// TIA Portal project "12_Converge_Station" (V19)

(* hardware
DEVICE "S7-1500/ET200MP station_1"  S7-1500 station
   slot 0: "Rail_0"  Rack  6ES7 590-1***0-0AA0
   slot 1: "PLC_1"  CPU 1513-1 PN  6ES7 513-1AL02-0AB0  V2.9
      slot 3: "CPU display_1"  6ES7591-1AA00-0AA0
      slot 32768: "PROFINET interface_1"  X1
         slot 32769: "Port_1"  X1 P1
         slot 32770: "Port_2"  X1 P2
      slot 34817: "Virtual CP interface port_1"  Virtual CP interface port  Virtual CP interface port
*)

// ===== PLC "PLC_1"  CPU 1513-1 PN =====

VAR_GLOBAL   // PLC tag table "Default tag table"
   "nw2" AT %M0.0 : Bool;
   "nw3 2nd memory (Pause)" AT %M0.2 : Bool;
   "nw3 1st memory (Unpause)" AT %M0.1 : Bool;
   "nw4" AT %M0.3 : Bool;
   "nw4 ae2 p" AT %M2.2 : Bool;
   "nw4 ae1 p" AT %M2.1 : Bool;
   "nw5" AT %M0.4 : Bool;
   "nw6 ae p" AT %M0.7 : Bool;
   "nw6" AT %M0.6 : Bool;
   "nw7 ae n" AT %M1.2 : Bool;
   "nw7" AT %M1.0 : Bool;
   "nw7 ae2 p" AT %M1.1 : Bool;
   "nw9 at2 p" AT %M1.7 : Bool;
   "nw9" AT %M1.6 : Bool;
   "nw9 at1 p" AT %M2.0 : Bool;
   "nw9 ae n" AT %M0.5 : Bool;
END_VAR

VAR_GLOBAL   // PLC tag table "Tag table from XML_1"
   "Start" AT %I0.0 : Bool;
   "Pause & Unpause" AT %I0.1 : Bool;
   "Reset" AT %I0.2 : Bool;
   "At entry 1" AT %I0.3 : Bool;
   "At transfer 1" AT %I0.4 : Bool;
   "At exit" AT %I0.5 : Bool;
   "At transfer 2" AT %I0.6 : Bool;
   "At entry 2" AT %I0.7 : Bool;
   "Auto" AT %I1.0 : Bool;
   "Manual" AT %I1.1 : Bool;
   "Start light" AT %Q0.0 : Bool;
   "P & UP light" AT %Q0.1 : Bool;
   "Reset light" AT %Q0.2 : Bool;
   "Load 1" AT %Q0.3 : Bool;
   "Load 2" AT %Q0.4 : Bool;
   "Transfer left 1" AT %Q0.5 : Bool;
   "Transfer left 2" AT %Q0.6 : Bool;
   "Conveyor 1" AT %Q0.7 : Bool;
   "Conveyor 2" AT %Q1.0 : Bool;
   "Exit conveyor" AT %Q1.1 : Bool;
   "Counter" AT %QD30 : DInt;
END_VAR

// folder: System blocks/Program resources

DATA_BLOCK "IEC_Counter_0_DB"   // DB1
{ S7_Optimized_Access := 'TRUE' }
AUTHOR : Simatic
FAMILY : IEC
NAME : CNTR
VERSION : 1.0
// stored: InstanceOfName IEC_COUNTER
"IEC_COUNTER"
BEGIN
END_DATA_BLOCK

// folder: (top level)

ORGANIZATION_BLOCK "Main"   // OB1, LAD, ProgramCycle
TITLE = "Main Program Sweep (Cycle)"
{ S7_Optimized_Access := 'TRUE' }
VERSION : 0.1
   VAR_INPUT
      Initial_Call : Bool;   // Initial call of this OB
      Remanence : Bool;   // =True, if remanent data are available
   END_VAR
   VAR_TEMP   // added for the SCL form of the ladder/FBD networks
      _w1 : Bool;
      _w2 : Bool;
   END_VAR
BEGIN

REGION Network 2: Start or Reset system with LED ON/OFF which are mounted on the switches
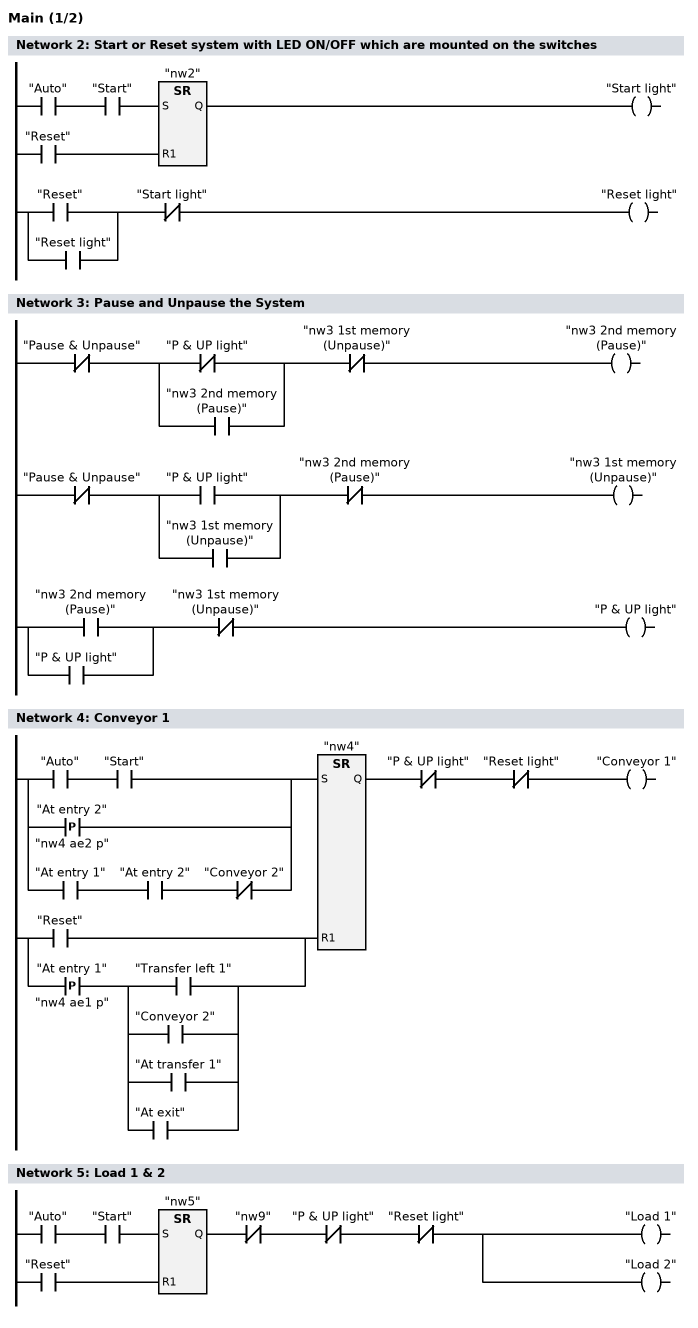
   RUNG wire#powerrail
      Contact( "Auto" )
      Contact( "Start" )
      S_SR(operand := "nw2", r1 := wire#w1)
      Coil( "Start light" )
   END_RUNG
   RUNG wire#powerrail
      Contact( "Reset" )
   END_RUNG wire#w1
   RUNG wire#powerrail
      Contact( "Reset" )
      wire#w2
      I_Contact( "Start light" )
      Coil( "Reset light" )
   END_RUNG
   RUNG wire#powerrail
      Contact( "Reset light" )
   END_RUNG wire#w2
   // the same network as SCL:
   IF "Auto" AND "Start" THEN
       "nw2" := TRUE;   // SR flip-flop
   END_IF;
   IF "Reset" THEN "nw2" := FALSE; END_IF;
   "Start light" := "nw2";
   "Reset light" := ("Reset" OR "Reset light") AND NOT "Start light";
END_REGION

REGION Network 3: Pause and Unpause the System
   RUNG wire#powerrail
      I_Contact( "Pause & Unpause" )
      wire#w1
      I_Contact( "P & UP light" )
      wire#w2
      I_Contact( "nw3 1st memory (Unpause)" )
      Coil( "nw3 2nd memory (Pause)" )
   END_RUNG
   RUNG wire#w1
      Contact( "nw3 2nd memory (Pause)" )
   END_RUNG wire#w2
   RUNG wire#powerrail
      I_Contact( "Pause & Unpause" )
      wire#w3
      Contact( "P & UP light" )
      wire#w4
      I_Contact( "nw3 2nd memory (Pause)" )
      Coil( "nw3 1st memory (Unpause)" )
   END_RUNG
   RUNG wire#w3
      Contact( "nw3 1st memory (Unpause)" )
   END_RUNG wire#w4
   RUNG wire#powerrail
      Contact( "nw3 2nd memory (Pause)" )
      wire#w5
      I_Contact( "nw3 1st memory (Unpause)" )
      Coil( "P & UP light" )
   END_RUNG
   RUNG wire#powerrail
      Contact( "P & UP light" )
   END_RUNG wire#w5
   // the same network as SCL:
   "nw3 2nd memory (Pause)" := NOT "Pause & Unpause" AND (NOT "P & UP light" OR "nw3 2nd memory (Pause)") AND NOT "nw3 1st memory (Unpause)";
   "nw3 1st memory (Unpause)" := NOT "Pause & Unpause" AND ("P & UP light" OR "nw3 1st memory (Unpause)") AND NOT "nw3 2nd memory (Pause)";
   "P & UP light" := ("nw3 2nd memory (Pause)" OR "P & UP light") AND NOT "nw3 1st memory (Unpause)";
END_REGION

REGION Network 4: Conveyor 1
   RUNG wire#powerrail
      Contact( "Auto" )
      Contact( "Start" )
      wire#w1
      S_SR(operand := "nw4", r1 := wire#w3)
      I_Contact( "P & UP light" )
      I_Contact( "Reset light" )
      Coil( "Conveyor 1" )
   END_RUNG
   RUNG wire#powerrail
      P_Contact(operand := "At entry 2", bit := "nw4 ae2 p")
   END_RUNG wire#w1
   RUNG wire#powerrail
      Contact( "At entry 1" )
      Contact( "At entry 2" )
      I_Contact( "Conveyor 2" )
   END_RUNG wire#w1
   RUNG wire#powerrail
      Contact( "Reset" )
   END_RUNG wire#w3
   RUNG wire#powerrail
      P_Contact(operand := "At entry 1", bit := "nw4 ae1 p")
      wire#w2
      Contact( "Transfer left 1" )
   END_RUNG wire#w3
   RUNG wire#w2
      Contact( "Conveyor 2" )
   END_RUNG wire#w3
   RUNG wire#w2
      Contact( "At transfer 1" )
   END_RUNG wire#w3
   RUNG wire#w2
      Contact( "At exit" )
   END_RUNG wire#w3
   // the same network as SCL:
   #_w1 := "At entry 2" AND NOT "nw4 ae2 p";   // rising edge of "At entry 2"
   "nw4 ae2 p" := "At entry 2";
   #_w2 := "At entry 1" AND NOT "nw4 ae1 p";   // rising edge of "At entry 1"
   "nw4 ae1 p" := "At entry 1";
   IF ("Auto" AND "Start") OR #_w1 OR ("At entry 1" AND "At entry 2" AND NOT "Conveyor 2") THEN
       "nw4" := TRUE;   // SR flip-flop
   END_IF;
   IF "Reset" OR (#_w2 AND ("Transfer left 1" OR "Conveyor 2" OR "At transfer 1" OR "At exit")) THEN
       "nw4" := FALSE;
   END_IF;
   "Conveyor 1" := "nw4" AND NOT "P & UP light" AND NOT "Reset light";
END_REGION

REGION Network 5: Load 1 & 2
   RUNG wire#powerrail
      Contact( "Auto" )
      Contact( "Start" )
      S_SR(operand := "nw5", r1 := wire#w1)
      I_Contact( "nw9" )
      I_Contact( "P & UP light" )
      I_Contact( "Reset light" )
      wire#w2
      Coil( "Load 1" )
   END_RUNG
   RUNG wire#powerrail
      Contact( "Reset" )
   END_RUNG wire#w1
   RUNG wire#w2
      Coil( "Load 2" )
   END_RUNG
   // the same network as SCL:
   IF "Auto" AND "Start" THEN
       "nw5" := TRUE;   // SR flip-flop
   END_IF;
   IF "Reset" THEN "nw5" := FALSE; END_IF;
   "Load 1" := "nw5" AND NOT "nw9" AND NOT "P & UP light" AND NOT "Reset light";
   "Load 2" := "Load 1";
END_REGION

REGION Network 6: Exit Conveyor in front of Conveyor 1
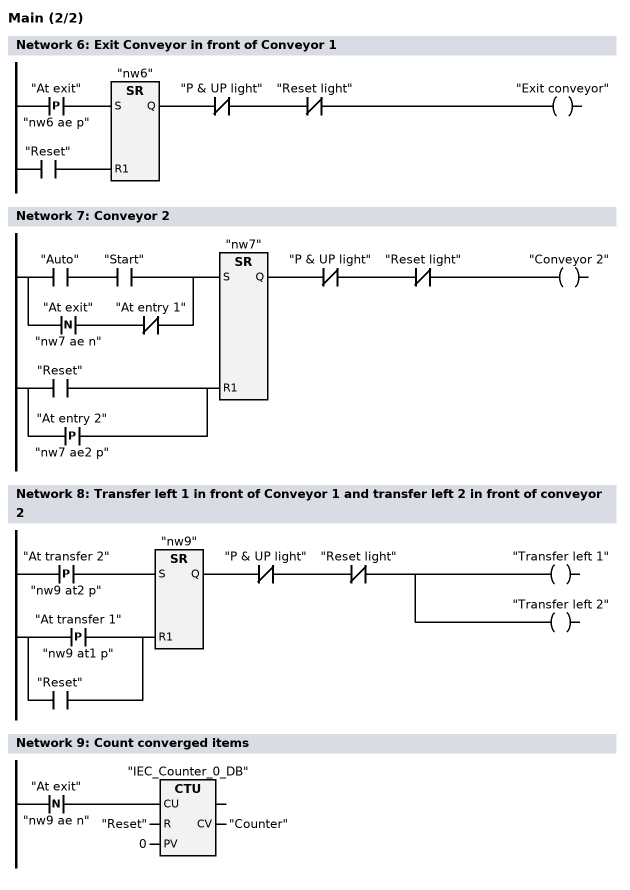
   RUNG wire#powerrail
      P_Contact(operand := "At exit", bit := "nw6 ae p")
      S_SR(operand := "nw6", r1 := wire#w1)
      I_Contact( "P & UP light" )
      I_Contact( "Reset light" )
      Coil( "Exit conveyor" )
   END_RUNG
   RUNG wire#powerrail
      Contact( "Reset" )
   END_RUNG wire#w1
   // the same network as SCL:
   #_w1 := "At exit" AND NOT "nw6 ae p";   // rising edge of "At exit"
   "nw6 ae p" := "At exit";
   IF #_w1 THEN
       "nw6" := TRUE;   // SR flip-flop
   END_IF;
   IF "Reset" THEN "nw6" := FALSE; END_IF;
   "Exit conveyor" := "nw6" AND NOT "P & UP light" AND NOT "Reset light";
END_REGION

REGION Network 7: Conveyor 2
   RUNG wire#powerrail
      Contact( "Auto" )
      Contact( "Start" )
      wire#w1
      S_SR(operand := "nw7", r1 := wire#w2)
      I_Contact( "P & UP light" )
      I_Contact( "Reset light" )
      Coil( "Conveyor 2" )
   END_RUNG
   RUNG wire#powerrail
      N_Contact(operand := "At exit", bit := "nw7 ae n")
      I_Contact( "At entry 1" )
   END_RUNG wire#w1
   RUNG wire#powerrail
      Contact( "Reset" )
   END_RUNG wire#w2
   RUNG wire#powerrail
      P_Contact(operand := "At entry 2", bit := "nw7 ae2 p")
   END_RUNG wire#w2
   // the same network as SCL:
   #_w1 := NOT "At exit" AND "nw7 ae n";   // falling edge of "At exit"
   "nw7 ae n" := "At exit";
   #_w2 := "At entry 2" AND NOT "nw7 ae2 p";   // rising edge of "At entry 2"
   "nw7 ae2 p" := "At entry 2";
   IF ("Auto" AND "Start") OR (#_w1 AND NOT "At entry 1") THEN
       "nw7" := TRUE;   // SR flip-flop
   END_IF;
   IF "Reset" OR #_w2 THEN "nw7" := FALSE; END_IF;
   "Conveyor 2" := "nw7" AND NOT "P & UP light" AND NOT "Reset light";
END_REGION

REGION Network 8: Transfer left 1 in front of Conveyor 1 and transfer left 2 in front of conveyor 2
   RUNG wire#powerrail
      P_Contact(operand := "At transfer 2", bit := "nw9 at2 p")
      S_SR(operand := "nw9", r1 := wire#w1)
      I_Contact( "P & UP light" )
      I_Contact( "Reset light" )
      wire#w2
      Coil( "Transfer left 1" )
   END_RUNG
   RUNG wire#powerrail
      P_Contact(operand := "At transfer 1", bit := "nw9 at1 p")
   END_RUNG wire#w1
   RUNG wire#powerrail
      Contact( "Reset" )
   END_RUNG wire#w1
   RUNG wire#w2
      Coil( "Transfer left 2" )
   END_RUNG
   // the same network as SCL:
   #_w1 := "At transfer 2" AND NOT "nw9 at2 p";   // rising edge of "At transfer 2"
   "nw9 at2 p" := "At transfer 2";
   #_w2 := "At transfer 1" AND NOT "nw9 at1 p";   // rising edge of "At transfer 1"
   "nw9 at1 p" := "At transfer 1";
   IF #_w1 THEN
       "nw9" := TRUE;   // SR flip-flop
   END_IF;
   IF #_w2 OR "Reset" THEN "nw9" := FALSE; END_IF;
   "Transfer left 1" := "nw9" AND NOT "P & UP light" AND NOT "Reset light";
   "Transfer left 2" := "Transfer left 1";
END_REGION

REGION Network 9: Count converged items
   #_w1 := NOT "At exit" AND "nw9 ae n";   // falling edge of "At exit"
   "nw9 ae n" := "At exit";
   "IEC_Counter_0_DB".CTU(CU := #_w1, R := "Reset", PV := 0, CV => "Counter");
END_REGION
END_ORGANIZATION_BLOCK